TEXTLIST TextList_06
   = ''
END_TEXTLIST

(* stored: Version 1.1.0.1
   TextList TextList_06: Id {2835816d-5859-0aae-0ceb-1d4dcd2c9b87} *)
